// TIA Portal V20 export
TYPE "LConSMC_typeMotionVector"
// stored: Access Published
   STRUCT
      s : LReal;   // [m] / [ft] Position
      v : LReal;   // [m/min] / [ft/min] Geschwindigkeit / [m/min] / [ft/min] Velocity
      "a" : LReal;   // [m/s^2] / [ft/s^2] Beschleunigung / [m/s^2] / [ft/s^2] Acceleration
   END_STRUCT;
END_TYPE
